(* Schneider Machine Expert - Basic project 友成插座（５个点）检测带２个安全门检测 - 副本 - 副本, file version 1.6.0.0 *)
(* ProjectInformations: Name=New project *)

HARDWARE
  Cpu 0: TM221CE40T
  EthernetConfiguration: NetworkName=M221, IpAllocationMode=FixedAddress, IpAddress=0.0.0.0, SubnetMask=0.0.0.0
  SerialLineConfiguration: Baud=Baud19200, Parity=ParityEven, DataBits=DataBits8, StopBits=StopBits1, PhysicalMedium=PhysicalMediumRs485, TransmissionMode=TransmissionModeModbusRtu, SlaveId=1, Addressing=SlaveAddressing
  MastTask: UsePeriodScanMode=false, PeriodScan=100
  FastTask: Period=255
  CpuBehavior: StartingMode=StartAsPreviousState, AutoSaveRamOnEeprom=true, WatchdogPeriod=250

SYMBOLS  (address, symbol, comment, settings)
  %M0         "左按钮"
  %M1         "右按钮"
  %M2         "拉料进到位感应"
  %M3         "伺服上限"
  %M4         "伺服中间感应位"
  %M5         "伺服下限"
  %M6         "机器安全门开关"
  %M7         "面板复位按扭"
  %M8         "面板停止按扭"
  %M9         "拉P汽缸到位"
  %M10        "導通1"
  %M11        "導通2"
  %M12        "導通3"
  %M13        "導通4"
  %M14        "導通5"
  %M15        "安全门检测位置"
  %M16        "安全门检测1"
  %M17        "安全门检测2"
  %M28        "暂停复位辅助"
  %M44        "拉p气缸向下辅助"
  %M45        "安全门测试电机向下辅助"
  %M46        "导通测试电机向下辅助"
  %M47        "执行拉P气缸动作"
  %M48        "执行安全门测试"
  %M49        "执行导通测试"
  %M50        "自动运行"
  %M51        "导通OK"
  %M52        "导通NG"
  %M53        "产品OK"
  %M54        "产品NG"
  %M55        "安全门打开复位辅助"
  %M102       "拉料气缸进"
  %M104       "双手启动按扭指示灯"
  %M105       "报警指示灯"
  %M106       "OK指示灯"
  %M107       "NG指示灯"
  %M108       "蜂鸣器"
  %M109       "拉料气缸出"
  %M110       "拉P汽缸"
  %M111       "拉P汽缸延時輔助"
  %M112       "上次第一次复位键有效"
  %M208       "复位完成"
  %M209       "电机向下"
  %M210       "电机向方向"
  %M213       "電機向上"
  %M215       "電機向下輔助"
  %S0       SB_COLDSTART  "Indicates or executes a cold start (data initialized to default values)"
  %S1       SB_WARMSTART  "Indicates there was a warm start with data backup"
  %S6       SB_TB1S  "Time base of 1 s generated by an internal clock"
  %S13      SB_FIRSTRUN  "Indicates the first controller cycle in RUN mode"
  %TM0        [Preset=5, Base=OneHundredMilliSeconds]
  %TM1        [Preset=5, Base=OneHundredMilliSeconds]
  %TM2        [Preset=2, Base=OneHundredMilliSeconds]
  %TM3        [Preset=2, Base=OneHundredMilliSeconds]
  %TM4        [Preset=5, Base=OneHundredMilliSeconds]
  %TM5        [Preset=5, Base=OneHundredMilliSeconds]
  %TM6        [Preset=5, Base=OneHundredMilliSeconds]
  %TM7        [Preset=2, Base=OneHundredMilliSeconds]
  %I0.0       "左按钮"
  %I0.1       "右按钮"
  %I0.2       "拉料进到位感应"
  %I0.3       "伺服上限"
  %I0.4       "伺服下限"
  %I0.5       "安全门检测位置"
  %I0.6       "机器安全门开关"
  %I0.7       "面板复位按扭"
  %I0.8       "面板停止按扭"
  %I0.9       "拉P汽缸到位"
  %I0.16      "安全门检测1"
  %I0.17      "安全门检测2"
  %Q0.1       "脉冲方向"
  %Q0.2       "拉料气缸进"
  %Q0.4       "双手启动按扭指示灯"
  %Q0.5       "报警指示灯"
  %Q0.6       "OK指示灯"
  %Q0.7       "NG指示灯"
  %Q0.8       "蜂鸣器"
  %Q0.9       "拉料气缸出"
  %Q0.10      "拉P汽缸"
  %Q0.11      "下顶"
  %PLS0       [PtoObject(RefInput=NotUsed, ZPhaseInput=NotUsed, ProbeInput=NotUsed), GlobalIndex=0, Type=PLS, TimeBase=ZeroPointOneMilliSeconds, Preset=1, UseDoubleWord=true]

POU 新 POU
  (* SectionNumber=1 *)

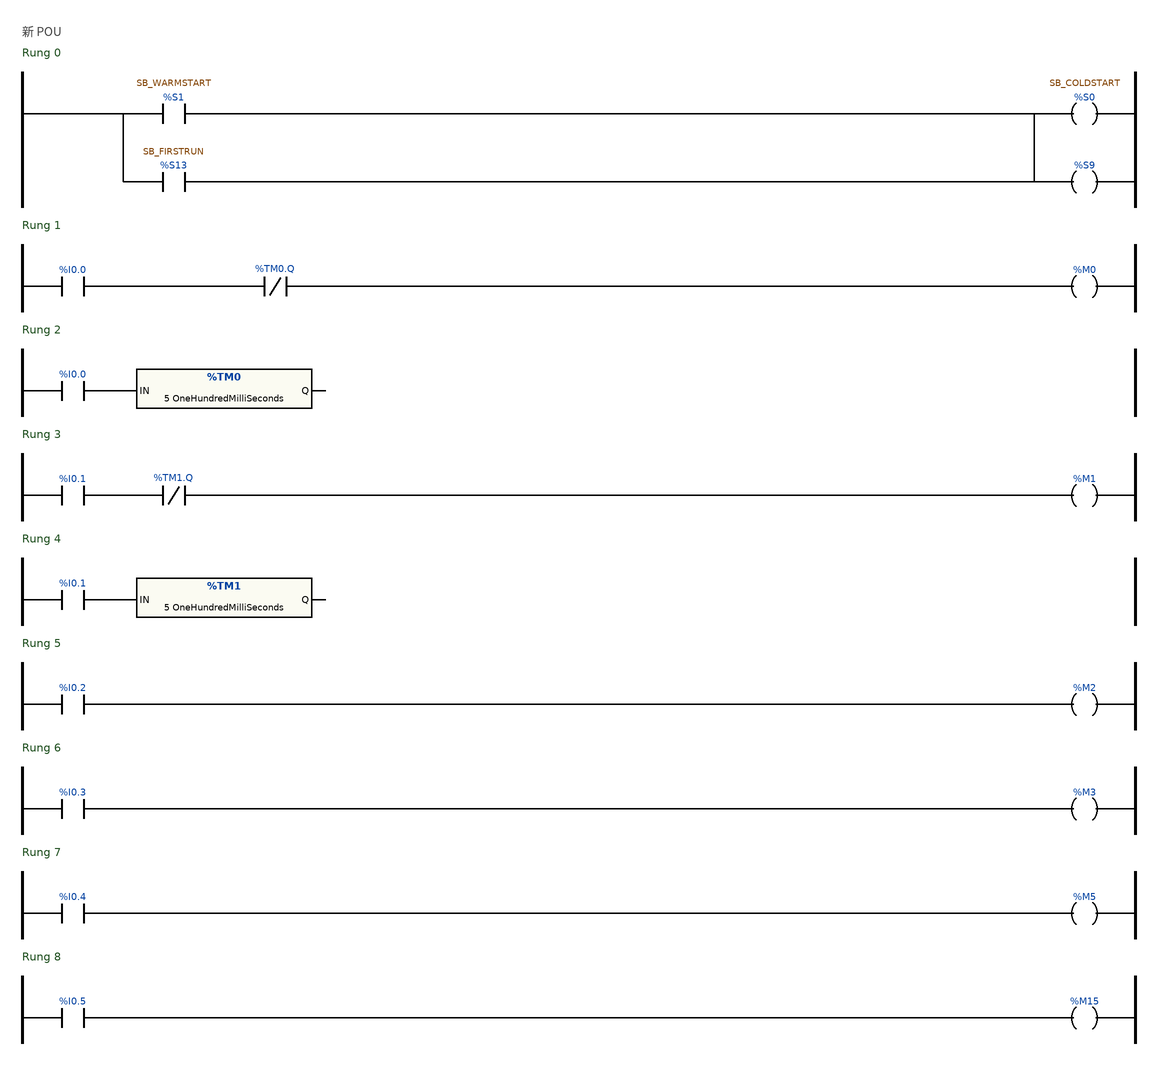

// Rung 0
  LD %S1                  (* SB_WARMSTART *)
  OR %S13                 (* SB_FIRSTRUN *)
  ST %S0                  (* SB_COLDSTART *)
  ST %S9
  // as ST:
  //   SB_COLDSTART := SB_WARMSTART OR SB_FIRSTRUN;
  //   %S9 := SB_WARMSTART OR SB_FIRSTRUN;

// Rung 1
  LD %I0.0
  ANDN %TM0.Q
  ST %M0
  // as ST:
  //   %M0 := %I0.0 AND NOT %TM0.Q;

// Rung 2
  BLK %TM0
  LD %I0.0
  IN
  END_BLK
  // as ST:
  //   %TM0(IN := %I0.0);

// Rung 3
  LD %I0.1
  ANDN %TM1.Q
  ST %M1
  // as ST:
  //   %M1 := %I0.1 AND NOT %TM1.Q;

// Rung 4
  BLK %TM1
  LD %I0.1
  IN
  END_BLK
  // as ST:
  //   %TM1(IN := %I0.1);

// Rung 5
  LD %I0.2
  ST %M2
  // as ST:
  //   %M2 := %I0.2;

// Rung 6
  LD %I0.3
  ST %M3
  // as ST:
  //   %M3 := %I0.3;

// Rung 7
  LD %I0.4
  ST %M5
  // as ST:
  //   %M5 := %I0.4;

// Rung 8
  LD %I0.5
  ST %M15
  // as ST:
  //   %M15 := %I0.5;

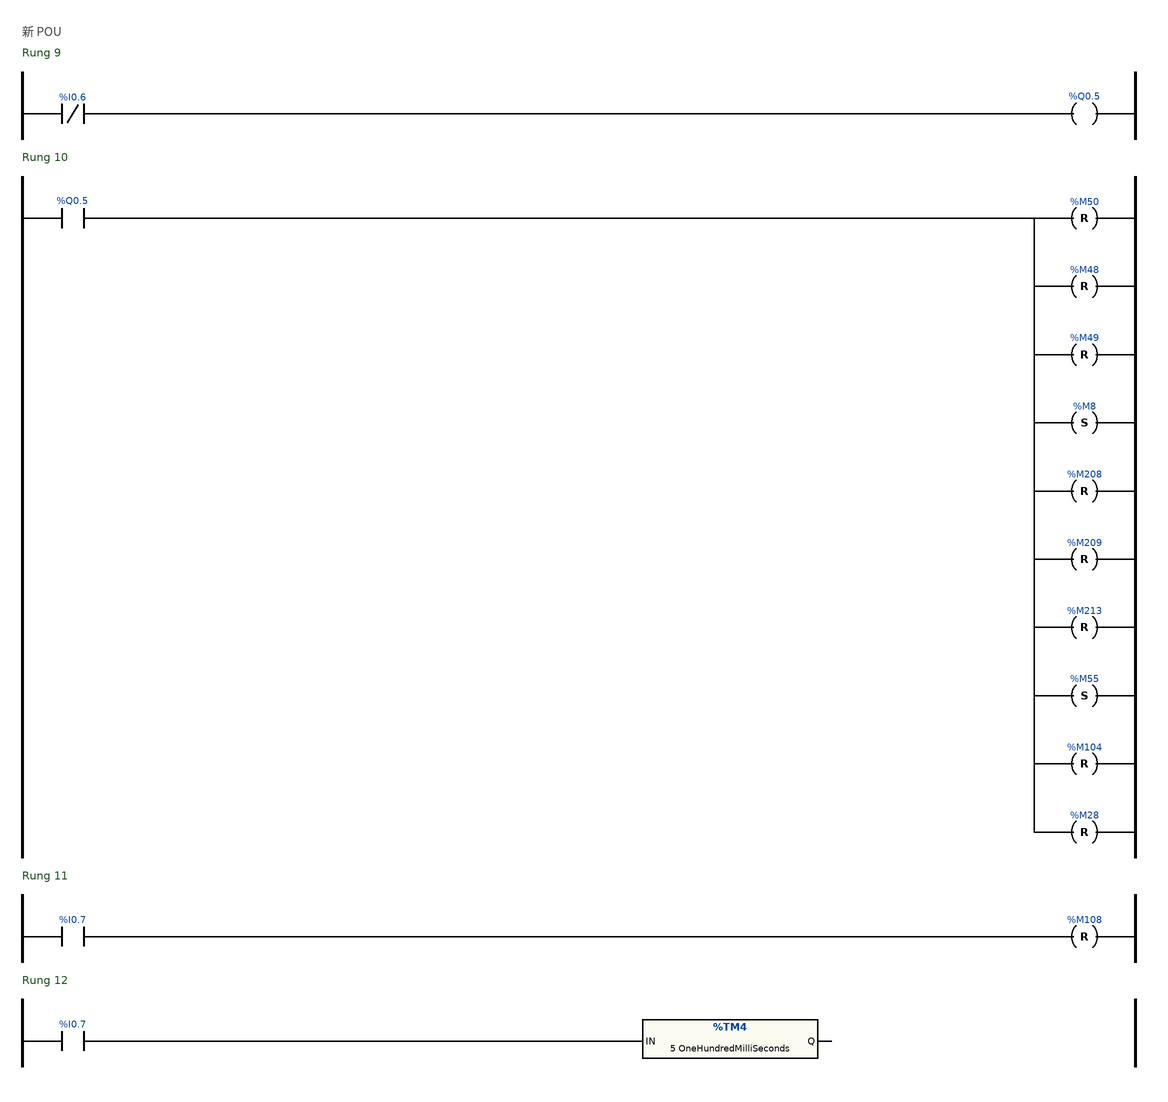

// Rung 9
  LDN %I0.6
  ST %Q0.5
  // as ST:
  //   %Q0.5 := NOT %I0.6;

// Rung 10
  LD %Q0.5
  R %M50
  R %M48
  R %M49
  S %M8
  R %M208
  R %M209
  R %M213
  S %M55
  R %M104
  R %M28
  // as ST:
  //   IF %Q0.5 THEN %M50 := FALSE; END_IF;
  //   IF %Q0.5 THEN %M48 := FALSE; END_IF;
  //   IF %Q0.5 THEN %M49 := FALSE; END_IF;
  //   IF %Q0.5 THEN %M8 := TRUE; END_IF;
  //   IF %Q0.5 THEN %M208 := FALSE; END_IF;
  //   IF %Q0.5 THEN %M209 := FALSE; END_IF;
  //   IF %Q0.5 THEN %M213 := FALSE; END_IF;
  //   IF %Q0.5 THEN %M55 := TRUE; END_IF;
  //   IF %Q0.5 THEN %M104 := FALSE; END_IF;
  //   IF %Q0.5 THEN %M28 := FALSE; END_IF;

// Rung 11
  LD %I0.7
  R %M108
  // as ST:
  //   IF %I0.7 THEN %M108 := FALSE; END_IF;

// Rung 12
  BLK %TM4
  LD %I0.7
  IN
  END_BLK
  // as ST:
  //   %TM4(IN := %I0.7);

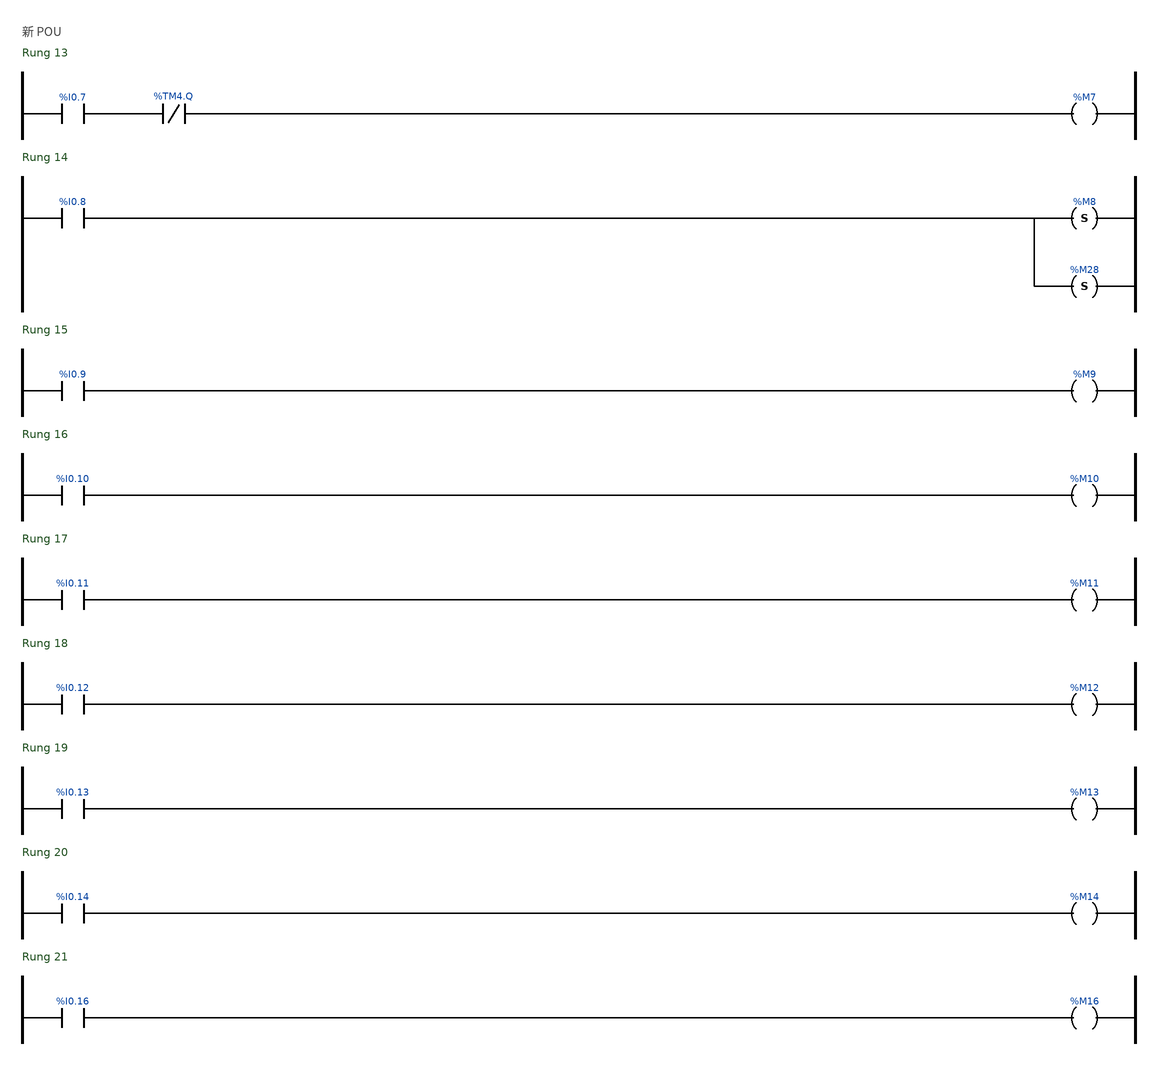

// Rung 13
  LD %I0.7
  ANDN %TM4.Q
  ST %M7
  // as ST:
  //   %M7 := %I0.7 AND NOT %TM4.Q;

// Rung 14
  LD %I0.8
  S %M8
  S %M28
  // as ST:
  //   IF %I0.8 THEN %M8 := TRUE; END_IF;
  //   IF %I0.8 THEN %M28 := TRUE; END_IF;

// Rung 15
  LD %I0.9
  ST %M9
  // as ST:
  //   %M9 := %I0.9;

// Rung 16
  LD %I0.10
  ST %M10
  // as ST:
  //   %M10 := %I0.10;

// Rung 17
  LD %I0.11
  ST %M11
  // as ST:
  //   %M11 := %I0.11;

// Rung 18
  LD %I0.12
  ST %M12
  // as ST:
  //   %M12 := %I0.12;

// Rung 19
  LD %I0.13
  ST %M13
  // as ST:
  //   %M13 := %I0.13;

// Rung 20
  LD %I0.14
  ST %M14
  // as ST:
  //   %M14 := %I0.14;

// Rung 21
  LD %I0.16
  ST %M16
  // as ST:
  //   %M16 := %I0.16;

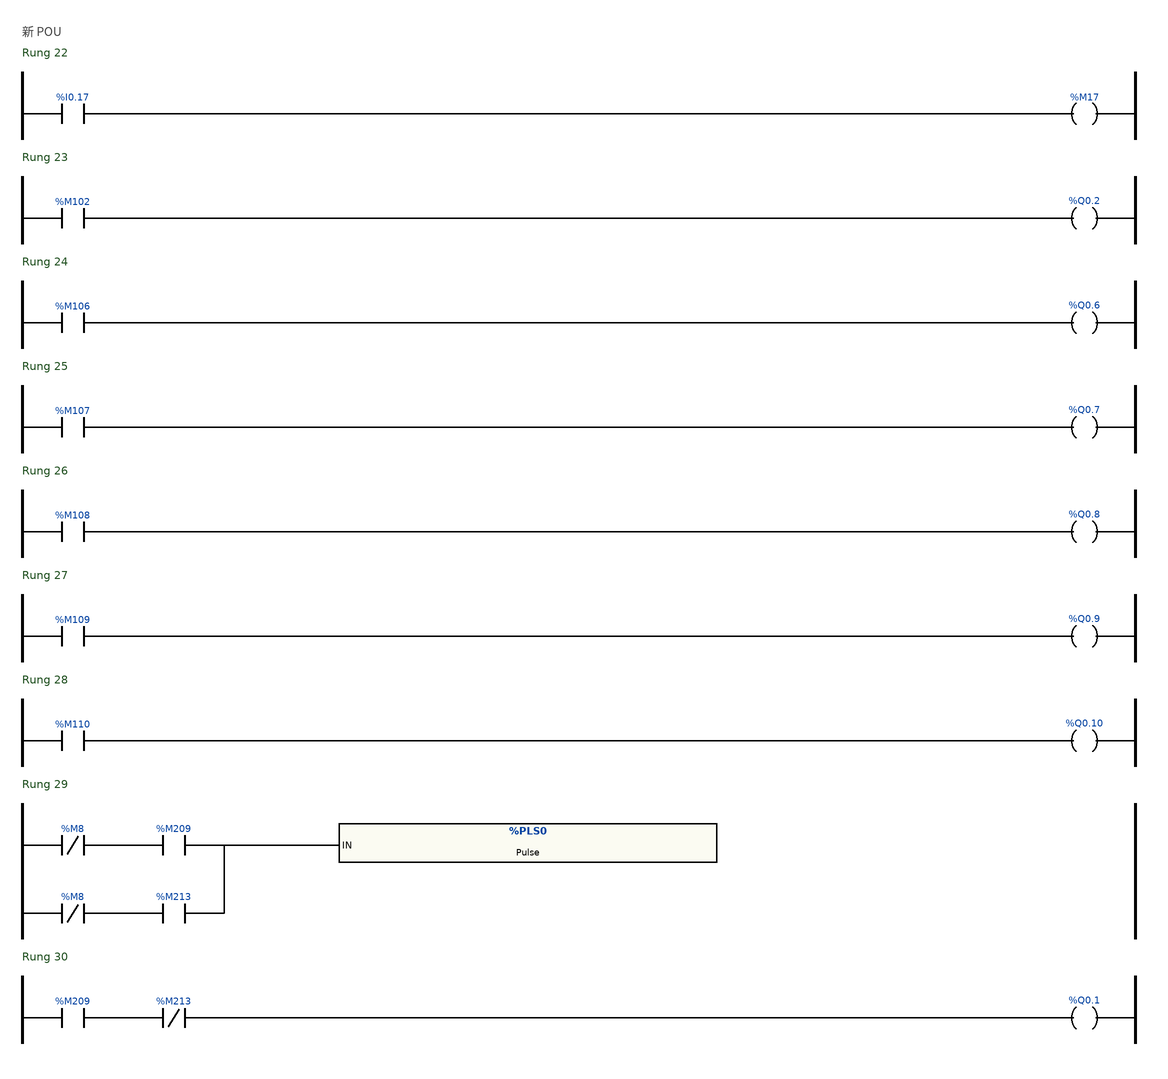

// Rung 22
  LD %I0.17
  ST %M17
  // as ST:
  //   %M17 := %I0.17;

// Rung 23
  LD %M102
  ST %Q0.2
  // as ST:
  //   %Q0.2 := %M102;

// Rung 24
  LD %M106
  ST %Q0.6
  // as ST:
  //   %Q0.6 := %M106;

// Rung 25
  LD %M107
  ST %Q0.7
  // as ST:
  //   %Q0.7 := %M107;

// Rung 26
  LD %M108
  ST %Q0.8
  // as ST:
  //   %Q0.8 := %M108;

// Rung 27
  LD %M109
  ST %Q0.9
  // as ST:
  //   %Q0.9 := %M109;

// Rung 28
  LD %M110
  ST %Q0.10
  // as ST:
  //   %Q0.10 := %M110;

// Rung 29
  BLK %PLS0
  LDN %M8
  AND %M209
  OR(N %M8
  AND %M213
  )
  IN
  END_BLK
  // as ST:
  //   %PLS0(IN := NOT %M8 AND %M209 OR NOT %M8 AND %M213);

// Rung 30
  LD %M209
  ANDN %M213
  ST %Q0.1
  // as ST:
  //   %Q0.1 := %M209 AND NOT %M213;

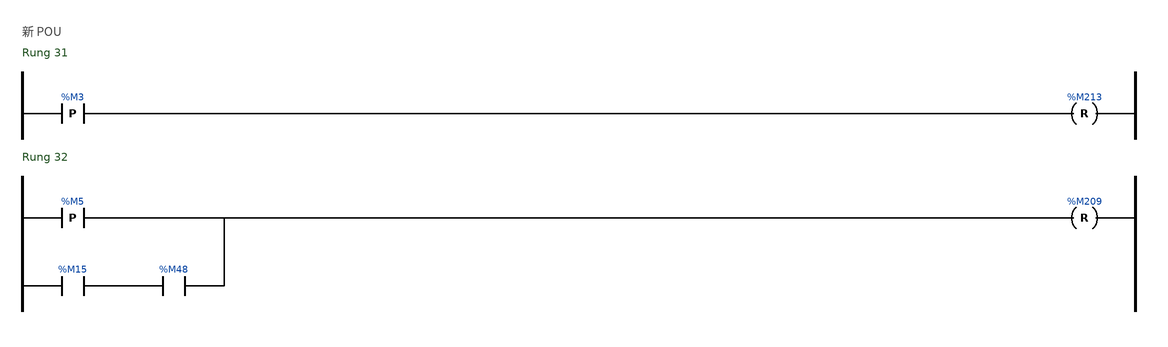

// Rung 31
  LDR %M3
  R %M213
  // as ST:
  //   IF RISING(%M3) THEN %M213 := FALSE; END_IF;

// Rung 32
  LDR %M5
  OR( %M15
  AND %M48
  )
  R %M209
  // as ST:
  //   IF RISING(%M5) OR %M15 AND %M48 THEN %M209 := FALSE; END_IF;

POU 新 POU
  (* SectionNumber=2 *)

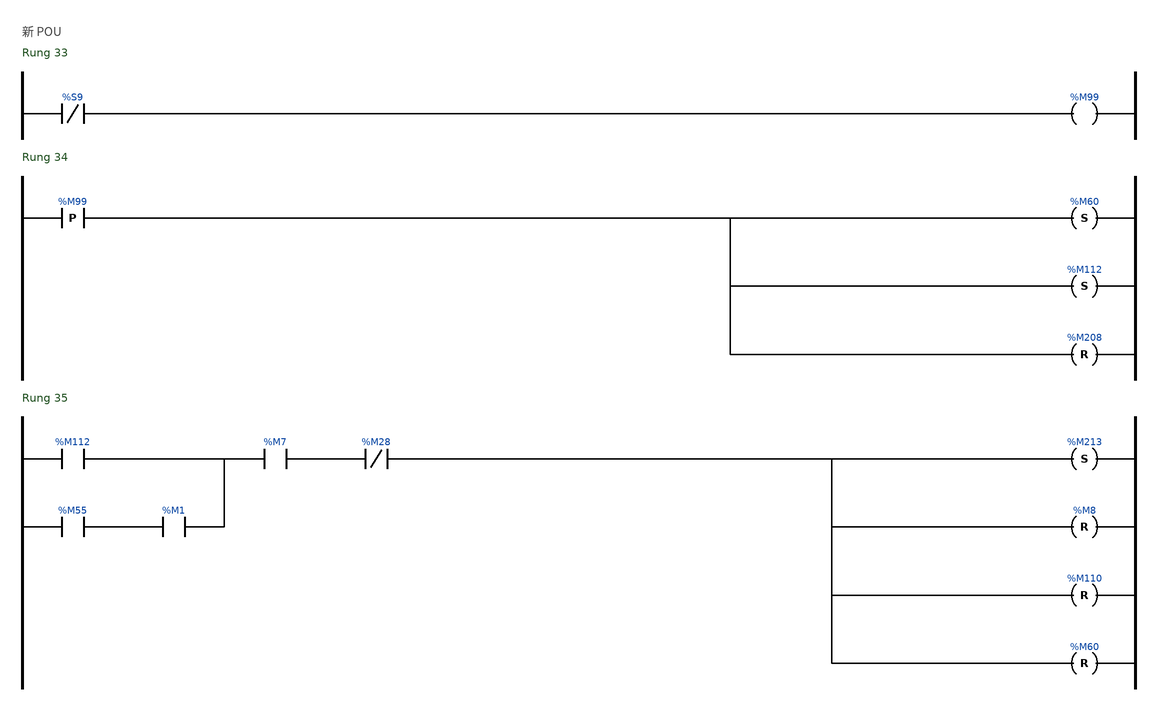

// Rung 33
  LDN %S9
  ST %M99
  // as ST:
  //   %M99 := NOT %S9;

// Rung 34
  LDR %M99
  S %M60
  S %M112
  R %M208
  // as ST:
  //   IF RISING(%M99) THEN %M60 := TRUE; END_IF;
  //   IF RISING(%M99) THEN %M112 := TRUE; END_IF;
  //   IF RISING(%M99) THEN %M208 := FALSE; END_IF;

// Rung 35
  LD %M112
  OR( %M55
  AND %M1
  )
  AND %M7
  ANDN %M28
  S %M213
  R %M8
  R %M110
  R %M60
  // as ST:
  //   IF (%M112 OR %M55 AND %M1) AND %M7 AND NOT %M28 THEN %M213 := TRUE; END_IF;
  //   IF (%M112 OR %M55 AND %M1) AND %M7 AND NOT %M28 THEN %M8 := FALSE; END_IF;
  //   IF (%M112 OR %M55 AND %M1) AND %M7 AND NOT %M28 THEN %M110 := FALSE; END_IF;
  //   IF (%M112 OR %M55 AND %M1) AND %M7 AND NOT %M28 THEN %M60 := FALSE; END_IF;

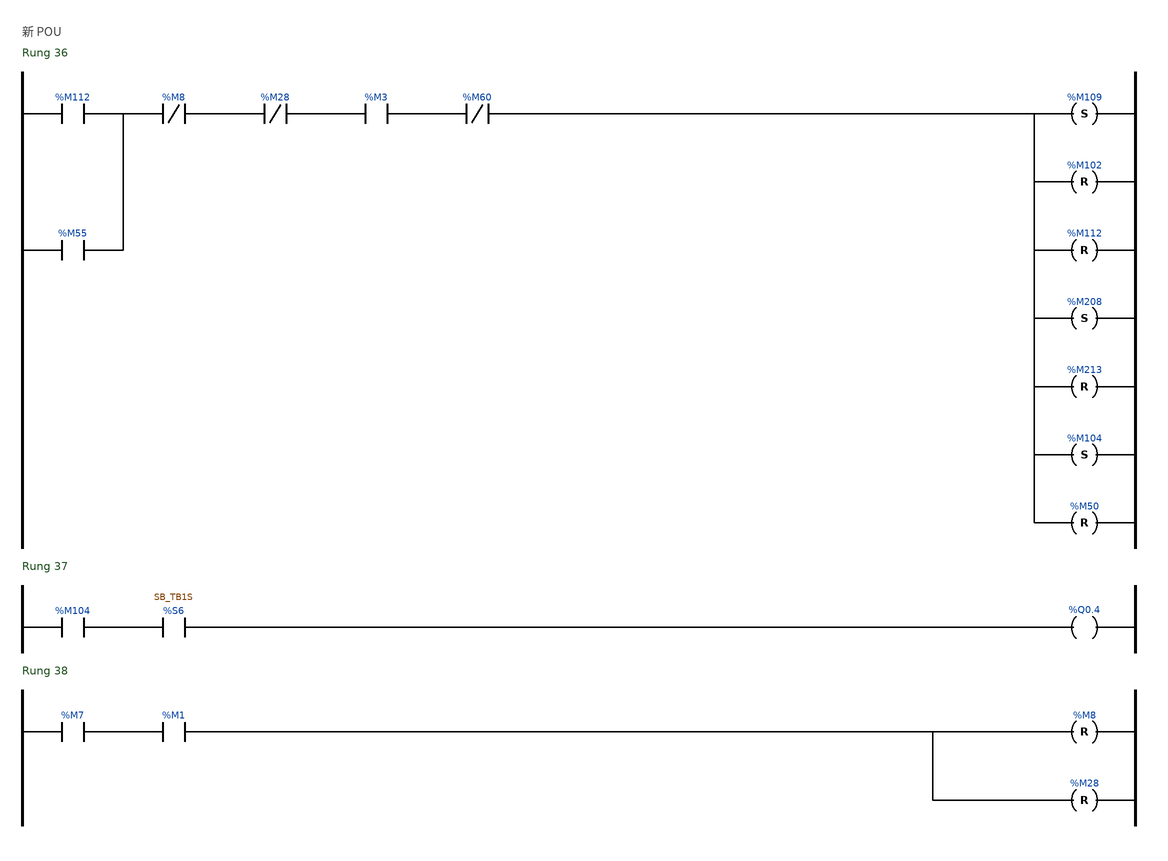

// Rung 36
  LD %M112
  OR %M55
  ANDN %M8
  ANDN %M28
  AND %M3
  ANDN %M60
  S %M109
  R %M102
  R %M112
  S %M208
  R %M213
  S %M104
  R %M50
  // as ST:
  //   IF (%M112 OR %M55) AND NOT %M8 AND NOT %M28 AND %M3 AND NOT %M60 THEN %M109 := TRUE; END_IF;
  //   IF (%M112 OR %M55) AND NOT %M8 AND NOT %M28 AND %M3 AND NOT %M60 THEN %M102 := FALSE; END_IF;
  //   _t1 := (%M112 OR %M55) AND NOT %M8 AND NOT %M28 AND %M3 AND NOT %M60;
  //   IF _t1 THEN %M112 := FALSE; END_IF;
  //   IF _t1 THEN %M208 := TRUE; END_IF;
  //   IF _t1 THEN %M213 := FALSE; END_IF;
  //   IF _t1 THEN %M104 := TRUE; END_IF;
  //   IF _t1 THEN %M50 := FALSE; END_IF;

// Rung 37
  LD %M104
  AND %S6                 (* SB_TB1S *)
  ST %Q0.4
  // as ST:
  //   %Q0.4 := %M104 AND SB_TB1S;

// Rung 38
  LD %M7
  AND %M1
  R %M8
  R %M28
  // as ST:
  //   IF %M7 AND %M1 THEN %M8 := FALSE; END_IF;
  //   IF %M7 AND %M1 THEN %M28 := FALSE; END_IF;

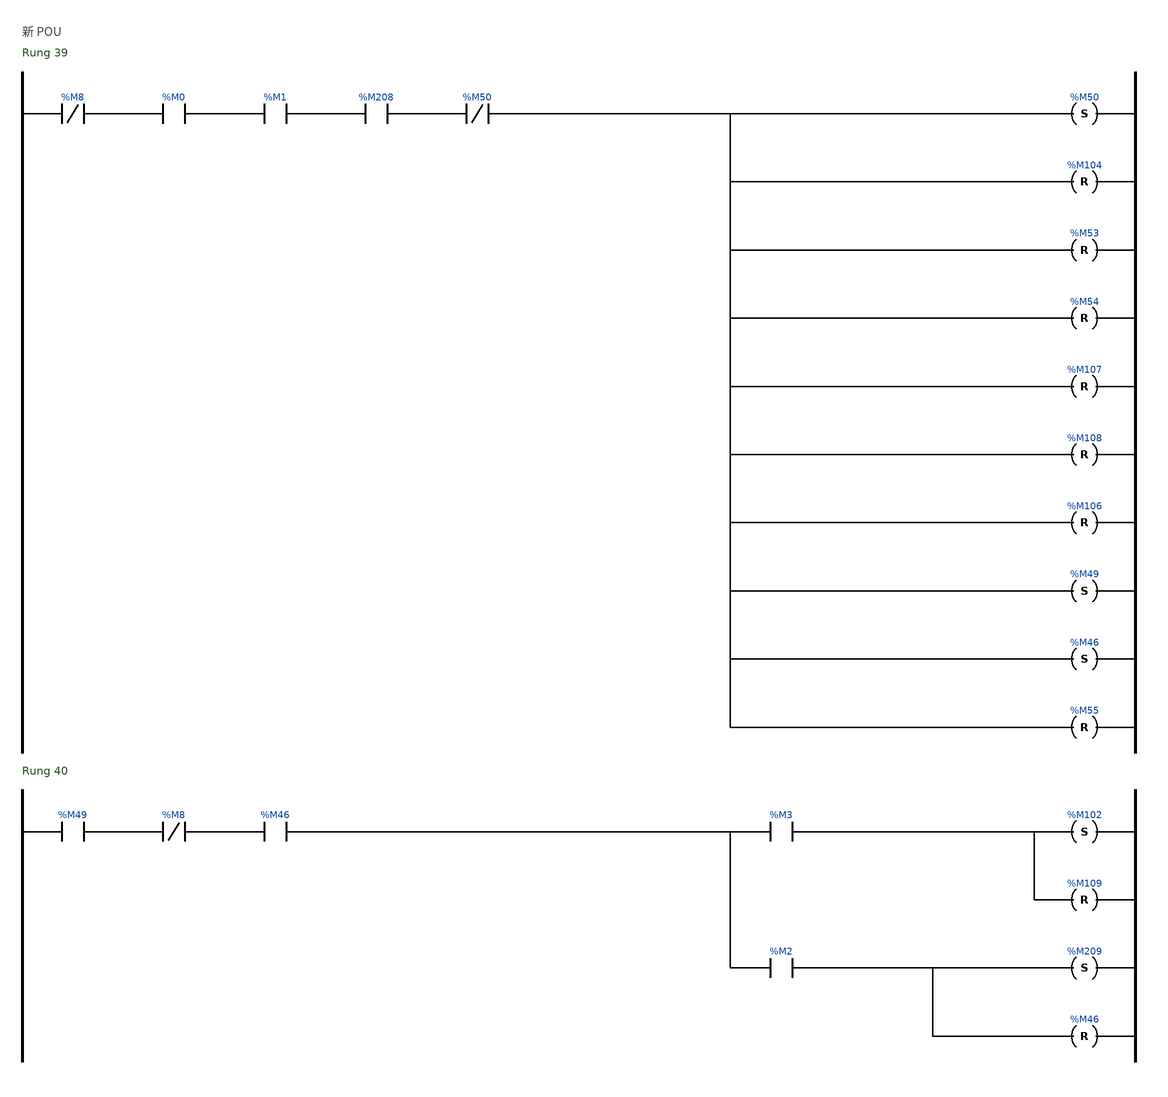

// Rung 39
  LDN %M8
  AND %M0
  AND %M1
  AND %M208
  ANDN %M50
  S %M50
  R %M104
  R %M53
  R %M54
  R %M107
  R %M108
  R %M106
  S %M49
  S %M46
  R %M55
  // as ST:
  //   _t1 := NOT %M8 AND %M0 AND %M1 AND %M208 AND NOT %M50;
  //   IF _t1 THEN %M50 := TRUE; END_IF;
  //   IF _t1 THEN %M104 := FALSE; END_IF;
  //   IF _t1 THEN %M53 := FALSE; END_IF;
  //   IF _t1 THEN %M54 := FALSE; END_IF;
  //   IF _t1 THEN %M107 := FALSE; END_IF;
  //   IF _t1 THEN %M108 := FALSE; END_IF;
  //   IF _t1 THEN %M106 := FALSE; END_IF;
  //   IF _t1 THEN %M49 := TRUE; END_IF;
  //   IF _t1 THEN %M46 := TRUE; END_IF;
  //   IF _t1 THEN %M55 := FALSE; END_IF;

// Rung 40
  LD %M49
  ANDN %M8
  AND %M46
  MPS
  AND %M3
  S %M102
  R %M109
  MPP
  AND %M2
  S %M209
  R %M46
  // as ST:
  //   IF %M49 AND NOT %M8 AND %M46 AND %M3 THEN %M102 := TRUE; END_IF;
  //   IF %M49 AND NOT %M8 AND %M46 AND %M3 THEN %M109 := FALSE; END_IF;
  //   IF %M49 AND NOT %M8 AND %M46 AND %M2 THEN %M209 := TRUE; END_IF;
  //   IF %M49 AND NOT %M8 AND %M46 AND %M2 THEN %M46 := FALSE; END_IF;

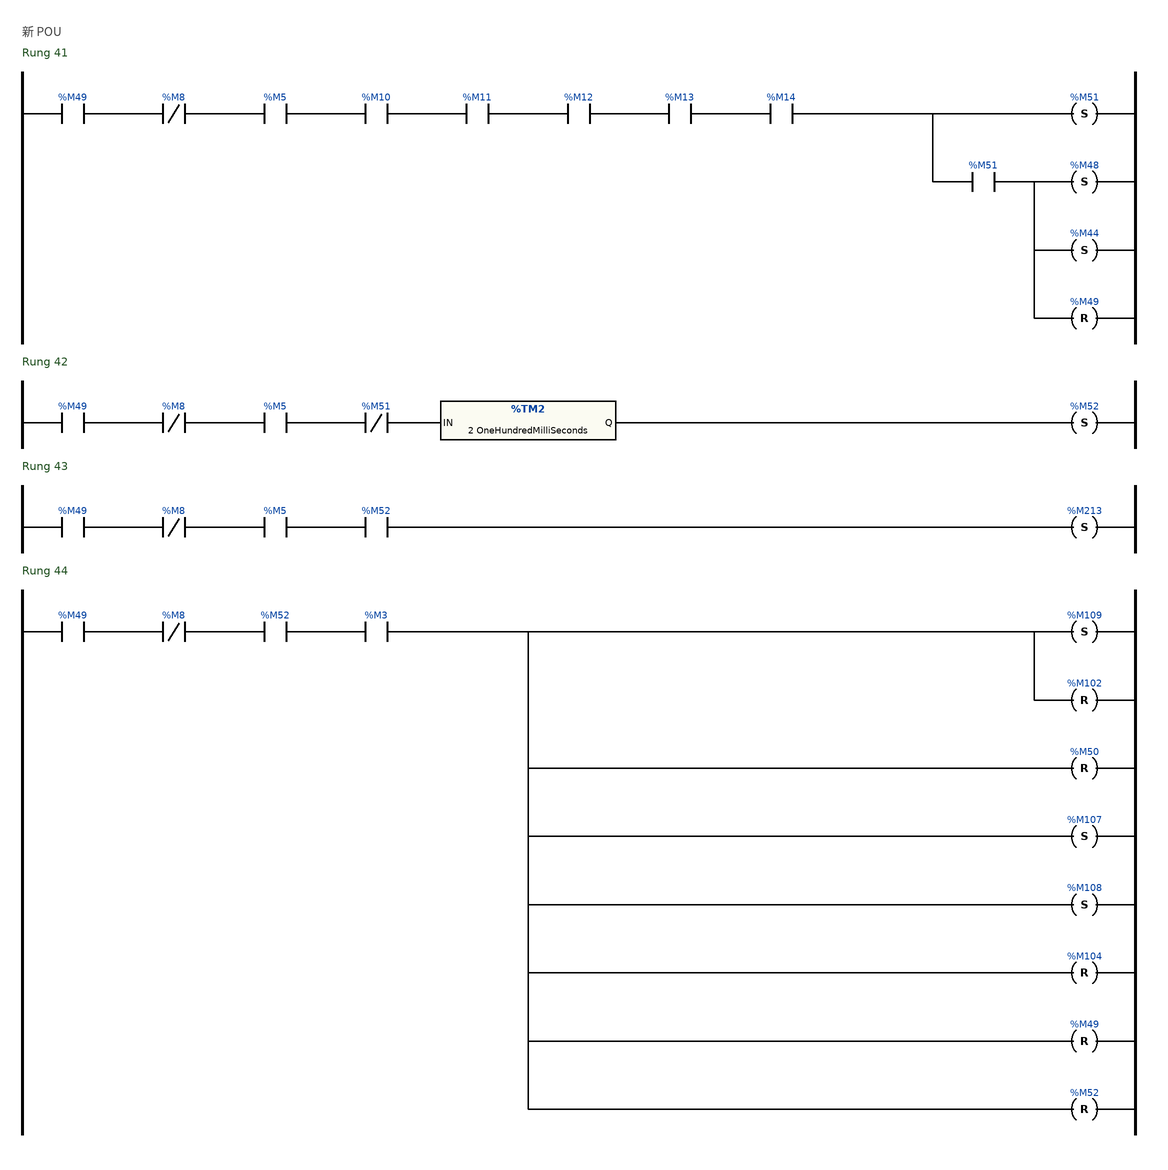

// Rung 41
  LD %M49
  ANDN %M8
  AND %M5
  AND %M10
  AND %M11
  AND %M12
  AND %M13
  AND %M14
  MPS
  S %M51
  MPP
  AND %M51
  S %M48
  S %M44
  R %M49
  // as ST:
  //   IF %M49 AND NOT %M8 AND %M5 AND %M10 AND %M11 AND %M12 AND %M13 AND %M14 THEN %M51 := TRUE; END_IF;
  //   IF %M49 AND NOT %M8 AND %M5 AND %M10 AND %M11 AND %M12 AND %M13 AND %M14 AND %M51 THEN %M48 := TRUE; END_IF;
  //   IF %M49 AND NOT %M8 AND %M5 AND %M10 AND %M11 AND %M12 AND %M13 AND %M14 AND %M51 THEN %M44 := TRUE; END_IF;
  //   IF %M49 AND NOT %M8 AND %M5 AND %M10 AND %M11 AND %M12 AND %M13 AND %M14 AND %M51 THEN %M49 := FALSE; END_IF;

// Rung 42
  BLK %TM2
  LD %M49
  ANDN %M8
  AND %M5
  ANDN %M51
  IN
  OUT_BLK
  LD Q
  S %M52
  END_BLK
  // as ST:
  //   %TM2(IN := %M49 AND NOT %M8 AND %M5 AND NOT %M51);
  //   IF %TM2.Q THEN %M52 := TRUE; END_IF;

// Rung 43
  LD %M49
  ANDN %M8
  AND %M5
  AND %M52
  S %M213
  // as ST:
  //   IF %M49 AND NOT %M8 AND %M5 AND %M52 THEN %M213 := TRUE; END_IF;

// Rung 44
  LD %M49
  ANDN %M8
  AND %M52
  AND %M3
  S %M109
  R %M102
  R %M50
  S %M107
  S %M108
  R %M104
  R %M49
  R %M52
  // as ST:
  //   IF %M49 AND NOT %M8 AND %M52 AND %M3 THEN %M109 := TRUE; END_IF;
  //   IF %M49 AND NOT %M8 AND %M52 AND %M3 THEN %M102 := FALSE; END_IF;
  //   IF %M49 AND NOT %M8 AND %M52 AND %M3 THEN %M50 := FALSE; END_IF;
  //   IF %M49 AND NOT %M8 AND %M52 AND %M3 THEN %M107 := TRUE; END_IF;
  //   IF %M49 AND NOT %M8 AND %M52 AND %M3 THEN %M108 := TRUE; END_IF;
  //   IF %M49 AND NOT %M8 AND %M52 AND %M3 THEN %M104 := FALSE; END_IF;
  //   _t1 := %M49 AND NOT %M8 AND %M52 AND %M3;
  //   IF _t1 THEN %M49 := FALSE; END_IF;
  //   IF _t1 THEN %M52 := FALSE; END_IF;

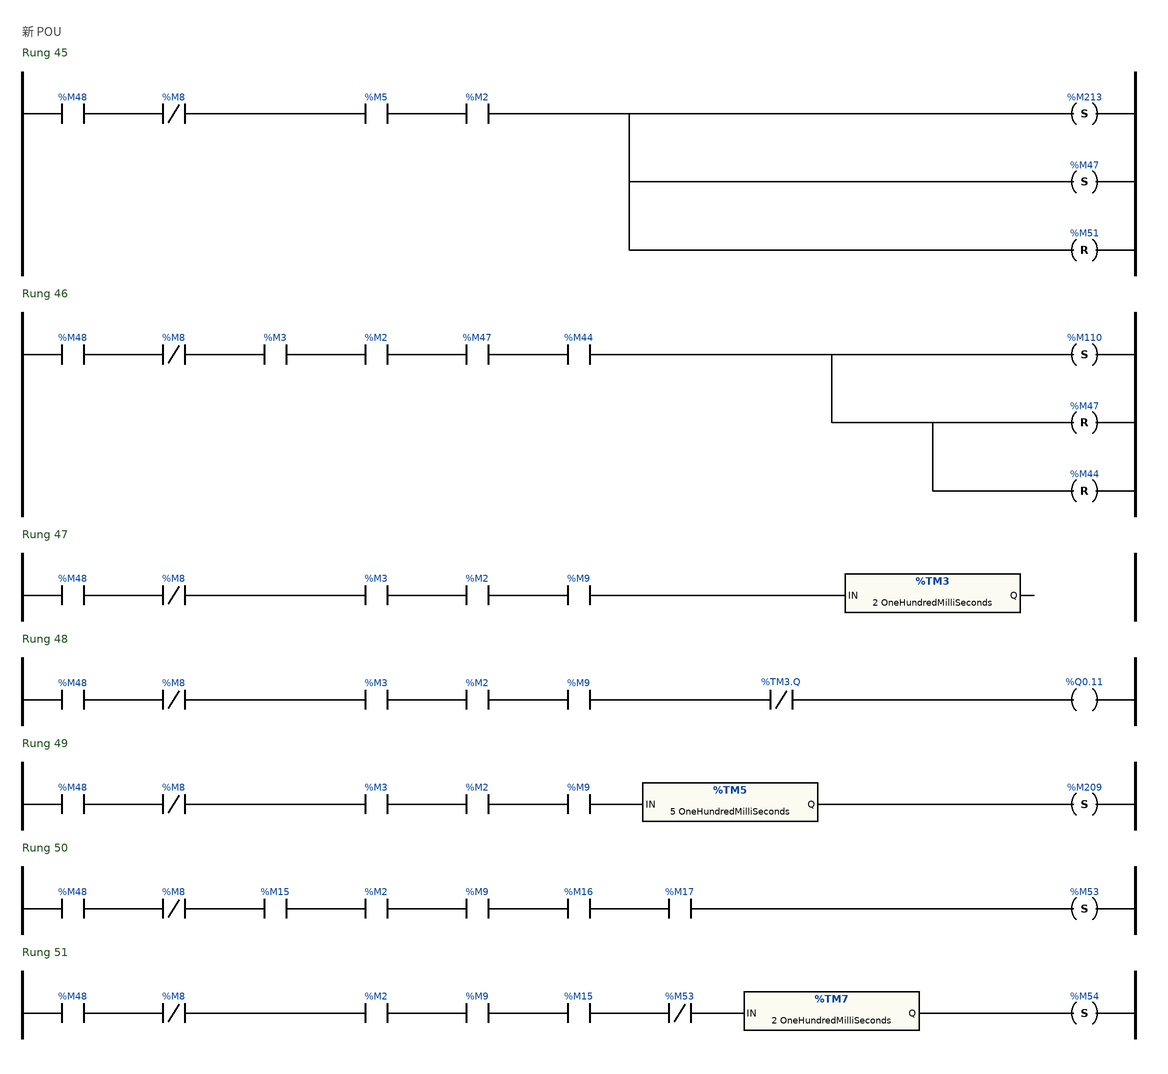

// Rung 45
  LD %M48
  ANDN %M8
  AND %M5
  AND %M2
  S %M213
  S %M47
  R %M51
  // as ST:
  //   IF %M48 AND NOT %M8 AND %M5 AND %M2 THEN %M213 := TRUE; END_IF;
  //   IF %M48 AND NOT %M8 AND %M5 AND %M2 THEN %M47 := TRUE; END_IF;
  //   IF %M48 AND NOT %M8 AND %M5 AND %M2 THEN %M51 := FALSE; END_IF;

// Rung 46
  LD %M48
  ANDN %M8
  AND %M3
  AND %M2
  AND %M47
  AND %M44
  S %M110
  R %M47
  R %M44
  // as ST:
  //   IF %M48 AND NOT %M8 AND %M3 AND %M2 AND %M47 AND %M44 THEN %M110 := TRUE; END_IF;
  //   _t1 := %M48 AND NOT %M8 AND %M3 AND %M2 AND %M47 AND %M44;
  //   IF _t1 THEN %M47 := FALSE; END_IF;
  //   IF _t1 THEN %M44 := FALSE; END_IF;

// Rung 47
  BLK %TM3
  LD %M48
  ANDN %M8
  AND %M3
  AND %M2
  AND %M9
  IN
  END_BLK
  // as ST:
  //   %TM3(IN := %M48 AND NOT %M8 AND %M3 AND %M2 AND %M9);

// Rung 48
  LD %M48
  ANDN %M8
  AND %M3
  AND %M2
  AND %M9
  ANDN %TM3.Q
  ST %Q0.11
  // as ST:
  //   %Q0.11 := %M48 AND NOT %M8 AND %M3 AND %M2 AND %M9 AND NOT %TM3.Q;

// Rung 49
  BLK %TM5
  LD %M48
  ANDN %M8
  AND %M3
  AND %M2
  AND %M9
  IN
  OUT_BLK
  LD Q
  S %M209
  END_BLK
  // as ST:
  //   %TM5(IN := %M48 AND NOT %M8 AND %M3 AND %M2 AND %M9);
  //   IF %TM5.Q THEN %M209 := TRUE; END_IF;

// Rung 50
  LD %M48
  ANDN %M8
  AND %M15
  AND %M2
  AND %M9
  AND %M16
  AND %M17
  S %M53
  // as ST:
  //   IF %M48 AND NOT %M8 AND %M15 AND %M2 AND %M9 AND %M16 AND %M17 THEN %M53 := TRUE; END_IF;

// Rung 51
  BLK %TM7
  LD %M48
  ANDN %M8
  AND %M2
  AND %M9
  AND %M15
  ANDN %M53
  IN
  OUT_BLK
  LD Q
  S %M54
  END_BLK
  // as ST:
  //   %TM7(IN := %M48 AND NOT %M8 AND %M2 AND %M9 AND %M15 AND NOT %M53);
  //   IF %TM7.Q THEN %M54 := TRUE; END_IF;

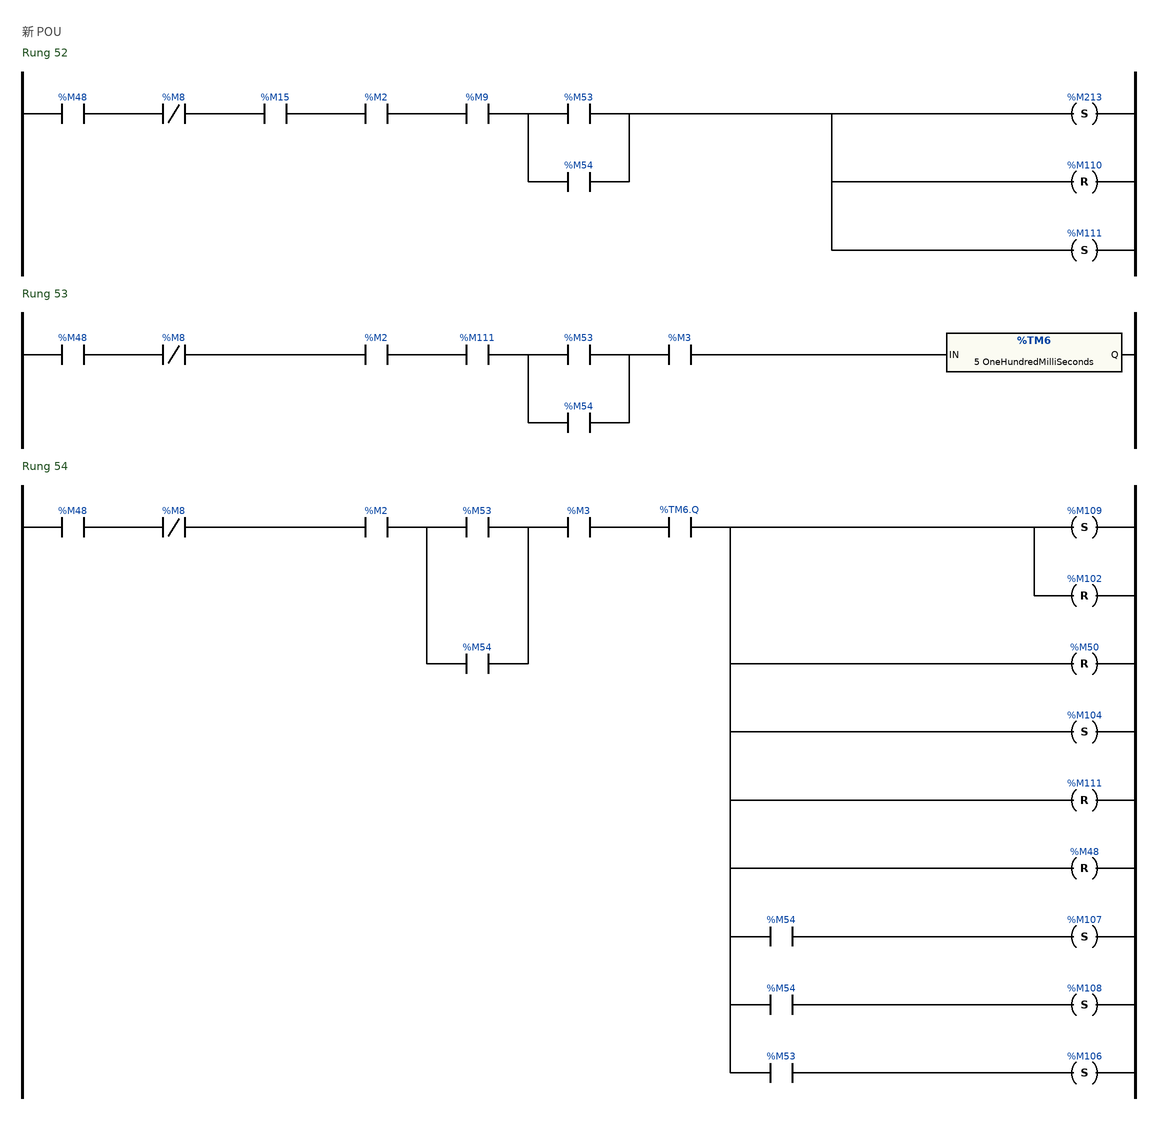

// Rung 52
  LD %M48
  ANDN %M8
  AND %M15
  AND %M2
  AND %M9
  AND( %M53
  OR %M54
  )
  S %M213
  R %M110
  S %M111
  // as ST:
  //   IF %M48 AND NOT %M8 AND %M15 AND %M2 AND %M9 AND (%M53 OR %M54) THEN %M213 := TRUE; END_IF;
  //   IF %M48 AND NOT %M8 AND %M15 AND %M2 AND %M9 AND (%M53 OR %M54) THEN %M110 := FALSE; END_IF;
  //   IF %M48 AND NOT %M8 AND %M15 AND %M2 AND %M9 AND (%M53 OR %M54) THEN %M111 := TRUE; END_IF;

// Rung 53
  BLK %TM6
  LD %M48
  ANDN %M8
  AND %M2
  AND %M111
  AND( %M53
  OR %M54
  )
  AND %M3
  IN
  END_BLK
  // as ST:
  //   %TM6(IN := %M48 AND NOT %M8 AND %M2 AND %M111 AND (%M53 OR %M54) AND %M3);

// Rung 54
  LD %M48
  ANDN %M8
  AND %M2
  AND( %M53
  OR %M54
  )
  AND %M3
  AND %TM6.Q
  MPS
  S %M109
  R %M102
  MRD
  R %M50
  MRD
  S %M104
  MRD
  R %M111
  MRD
  R %M48
  MRD
  AND %M54
  S %M107
  MRD
  AND %M54
  S %M108
  MPP
  AND %M53
  S %M106
  // as ST:
  //   IF %M48 AND NOT %M8 AND %M2 AND (%M53 OR %M54) AND %M3 AND %TM6.Q THEN %M109 := TRUE; END_IF;
  //   IF %M48 AND NOT %M8 AND %M2 AND (%M53 OR %M54) AND %M3 AND %TM6.Q THEN %M102 := FALSE; END_IF;
  //   IF %M48 AND NOT %M8 AND %M2 AND (%M53 OR %M54) AND %M3 AND %TM6.Q THEN %M50 := FALSE; END_IF;
  //   IF %M48 AND NOT %M8 AND %M2 AND (%M53 OR %M54) AND %M3 AND %TM6.Q THEN %M104 := TRUE; END_IF;
  //   IF %M48 AND NOT %M8 AND %M2 AND (%M53 OR %M54) AND %M3 AND %TM6.Q THEN %M111 := FALSE; END_IF;
  //   _t1 := %M48 AND NOT %M8 AND %M2 AND (%M53 OR %M54) AND %M3 AND %TM6.Q;
  //   IF _t1 THEN %M48 := FALSE; END_IF;
  //   IF _t1 AND %M54 THEN %M107 := TRUE; END_IF;
  //   IF _t1 AND %M54 THEN %M108 := TRUE; END_IF;
  //   IF _t1 AND %M53 THEN %M106 := TRUE; END_IF;
